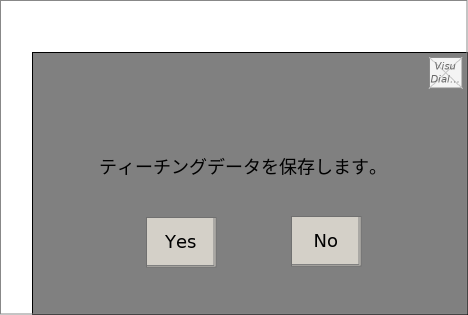
VISUALIZATION d_gm_saveBtn  // 468x315
    Rectangle (32,52 436x263)
    Image (429,57 33x31), image: VisuDialogs.ImagePoolDialogs.Delete
        OnMouseClick: CloseDialog Dialog=d_gm_saveBtn, Result=OK, NumpadKeypadSet=True
    Label (56,140 374x55), "ティーチングデータを保存します。"
    Button (146,217 70x50), "Yes"
        tap gvl_visu.flg_btn_rotaryPos
        OnMouseClick: CloseDialog Dialog=d_gm_saveBtn, Result=OK, NumpadKeypadSet=True
    Button (291,216 70x50), "No"
        OnMouseClick: CloseDialog Dialog=d_gm_saveBtn, Result=OK, NumpadKeypadSet=True
END_VISUALIZATION

(* stored: Version 1.1.0.1, ProductVersion 3.1.4024.12
   Visu d_gm_saveBtn: Id {011ede35-f9a2-4613-b413-051af3ce0304} *)
